FUNCTION_BLOCK FB_Marquee
VAR_INPUT
	pLamp01			:POINTER TO BOOL;
	pLamp02			:POINTER TO BOOL;
	pLamp03			:POINTER TO BOOL;
	pLamp04			:POINTER TO BOOL;
END_VAR
VAR_OUTPUT
END_VAR
VAR
	TON1		:TON;
	TON2		:TON;
	TON3		:TON;
	TON4		:TON;
	rTrig		:F_TRIG;
	iStep		:INT;
END_VAR

METHOD Blinking : BOOL
VAR_INPUT
	bStart			:BOOL;
END_VAR
(*IF bStart THEN
	 
	TON1(IN:=TRUE, PT:= T#1S, Q=> , ET=> );
	pLamp01^ := TRUE;
	
	IF	TON1.Q THEN 
		pLamp01^ := FALSE;
		TON2(IN:=TON1.Q, PT:= T#1S, Q=> , ET=> );
		pLamp02^ := TRUE;
		IF TON2.Q THEN 
			pLamp02^ := FALSE;
			TON3(IN:=TON2.Q, PT:= T#1S, Q=> , ET=> );
			pLamp03^ := TRUE;
			IF TON3.Q THEN 
				pLamp03^ := FALSE;
				TON4(IN:=TON3.Q, PT:= T#1S, Q=> , ET=> );
				pLamp04^ := TRUE;
				IF TON4.Q THEN 
					pLamp04^ := FALSE;
					TON1(IN:=FALSE);
					
				END_IF
			END_IF
		END_IF
	END_IF *)
	
IF bStart THEN 
	CASE iStep OF
			0:
				pLamp01^ := TRUE;
				TON1(IN:=TRUE, PT:= T#1S, Q=> , ET=> );
				IF TON1.Q THEN 
					pLamp01^ := FALSE;
					TON1(IN:=FALSE);
					iStep:= 10;
				END_IF
			10:
				pLamp02^ := TRUE;
				TON2(IN:=TRUE, PT:=T#1S, Q=> , ET=> );
				IF TON2.Q THEN 
					pLamp02^ := FALSE;
					TON2(IN:=FALSE);
					iStep := 20;				
				END_IF
			20:
				pLamp03^ := TRUE;
				TON3(IN:=TRUE, PT:=T#1S, Q=> , ET=> );
				IF TON3.Q THEN 
					pLamp03^ := FALSE;
					TON3(IN:=FALSE);
					iStep := 30;
				END_IF
			30:
				pLamp04^ := TRUE;
				TON4(IN:=TRUE, PT:=T#1S, Q=> , ET=> );
				IF	TON4.Q THEN 
					pLamp04^ := FALSE;
					TON4(IN:=FALSE);
					iStep := 0;
				END_IF
	END_CASE
ELSE 
	pLamp04^ := FALSE;
	pLamp03^ := FALSE;
	pLamp02^ := FALSE;
	pLamp01^ := FALSE;
END_IF
END_METHOD

END_FUNCTION_BLOCK

(* stored: Version 1.1.0.1, ProductVersion 3.1.4022.16
   POU FB_Marquee: Id {ffdf7d82-b4ab-4511-9b34-b7a7860a4a5b}, SpecialFunc None
   Method Blinking: Id {d75e3a2d-b19b-4822-b107-2b2360cead3b} *)
